{attribute 'no_explicit_call' := 'NormallyOpenPushButton is a CLASS and must be accessed using methods or properties'}
FUNCTION_BLOCK NormallyOpenPushButton implements I_PushButton
VAR
	input				AT %I*: BOOL;
END_VAR

PROPERTY IsPressed : bool
GET
IsPressed				:= input;
END_GET
END_PROPERTY

PROPERTY IsReleased : bool
GET
IsReleased				:= not input;
END_GET
END_PROPERTY

END_FUNCTION_BLOCK

(* stored: Version 1.1.0.1, ProductVersion 3.1.4024.11
   POU NormallyOpenPushButton: Id {a96c7336-46b7-420c-8fa7-8d8ccfdc5b62}, SpecialFunc None
   Property IsPressed: Id {108eca65-6af9-46c3-b96d-8fbc1204f132}
   Get Get: Id {4376b41e-abdf-4d02-b41c-c33111fe5e53}
   Property IsReleased: Id {ba1f13f1-76f1-4cd6-abb0-08e8e76c2e5d}
   Get Get: Id {d0a958e4-495b-4d29-bb29-f6ddce91e6ac} *)
